% RSLogix 500 project Inventory_Management.RSS, saved by version 8.30.00.16 %
PROJECT "UNTITLED"    % processor: Bul.1763 MicroLogix 1100 Series B %

PROGRAM FILES
  LAD 2   9 rungs

DATA FILES
  O0 OUTPUT  4 elements
  I1 INPUT  6 elements
  S2 STATUS  66 elements
  B3 BINARY  1 elements
  T4 TIMER  1 elements
  C5 COUNTER  1 elements
  R6 CONTROL  1 elements
  N7 INTEGER  4 elements
  F8 FLOAT  1 elements
  ST9 STRING  10 elements

LADDER 2
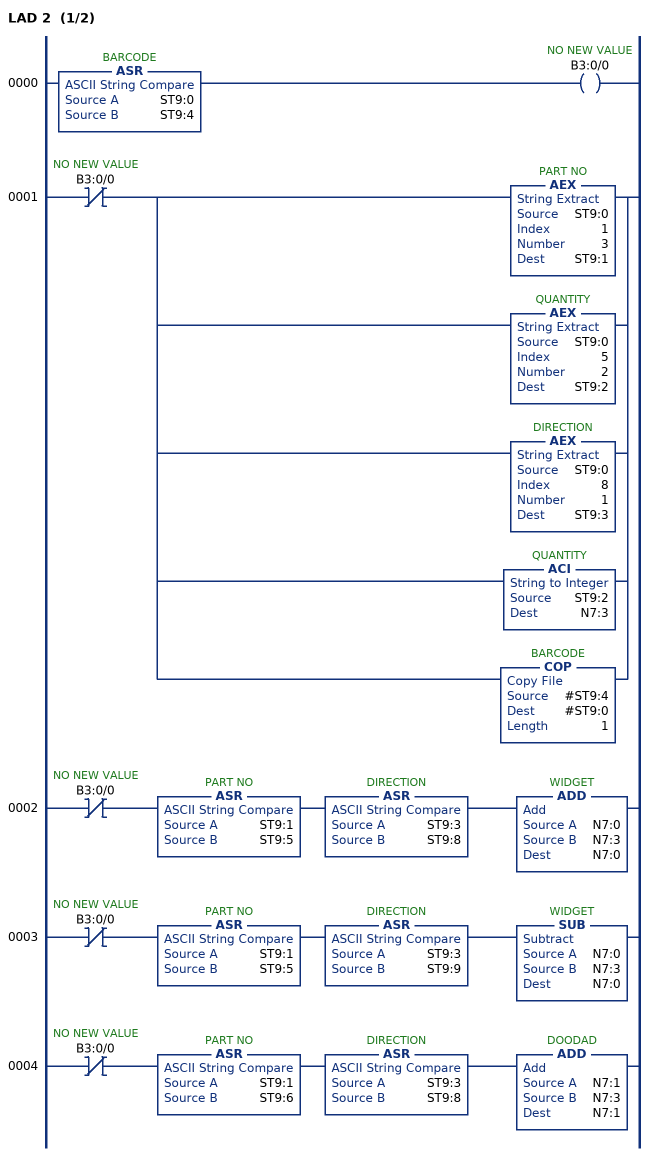
% Rung: 0 %
SOR ASR ST9:0 ST9:4 OTE B3:0/0 EOR
%   ST9:0  "BARCODE" %
%   B3:0/0  "NO NEW VALUE" %
% Rung: 1 %
SOR XIO B3:0/0 BST AEX ST9:0 1 3 ST9:1 NXB AEX ST9:0 5 2 ST9:2 NXB AEX ST9:0 8 1 ST9:3 NXB ACI ST9:2 N7:3 NXB COP #ST9:4 #ST9:0 1 BND EOR
%   B3:0/0  "NO NEW VALUE" %
%   ST9:0  "BARCODE" %
%   ST9:1  "PART NO" %
%   ST9:2  "QUANTITY" %
%   ST9:3  "DIRECTION" %
%   N7:3  "QUANTITY" %
% Rung: 2 %
SOR XIO B3:0/0 ASR ST9:1 ST9:5 ASR ST9:3 ST9:8 ADD N7:0 N7:3 N7:0 EOR
%   B3:0/0  "NO NEW VALUE" %
%   ST9:1  "PART NO" %
%   ST9:3  "DIRECTION" %
%   N7:0  "WIDGET" %
%   N7:3  "QUANTITY" %
% Rung: 3 %
SOR XIO B3:0/0 ASR ST9:1 ST9:5 ASR ST9:3 ST9:9 SUB N7:0 N7:3 N7:0 EOR
%   B3:0/0  "NO NEW VALUE" %
%   ST9:1  "PART NO" %
%   ST9:3  "DIRECTION" %
%   N7:0  "WIDGET" %
%   N7:3  "QUANTITY" %
% Rung: 4 %
SOR XIO B3:0/0 ASR ST9:1 ST9:6 ASR ST9:3 ST9:8 ADD N7:1 N7:3 N7:1 EOR
%   B3:0/0  "NO NEW VALUE" %
%   ST9:1  "PART NO" %
%   ST9:6  "PART NO" %
%   ST9:3  "DIRECTION" %
%   N7:1  "DOODAD" %
%   N7:3  "QUANTITY" %

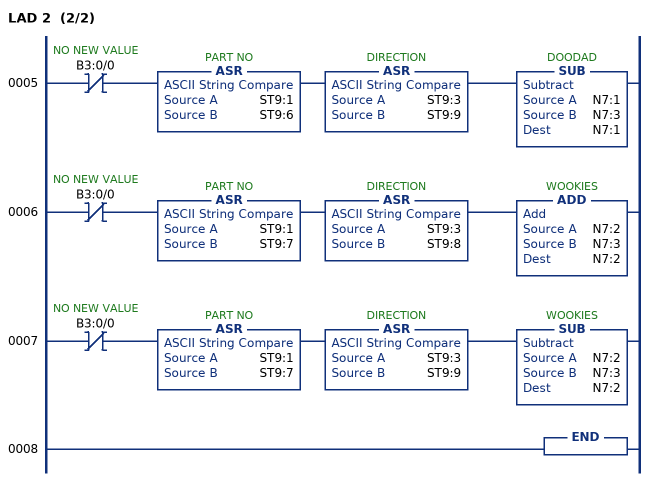
% Rung: 5 %
SOR XIO B3:0/0 ASR ST9:1 ST9:6 ASR ST9:3 ST9:9 SUB N7:1 N7:3 N7:1 EOR
%   B3:0/0  "NO NEW VALUE" %
%   ST9:1  "PART NO" %
%   ST9:6  "PART NO" %
%   ST9:3  "DIRECTION" %
%   N7:1  "DOODAD" %
%   N7:3  "QUANTITY" %
% Rung: 6 %
SOR XIO B3:0/0 ASR ST9:1 ST9:7 ASR ST9:3 ST9:8 ADD N7:2 N7:3 N7:2 EOR
%   B3:0/0  "NO NEW VALUE" %
%   ST9:1  "PART NO" %
%   ST9:3  "DIRECTION" %
%   N7:2  "WOOKIES" %
%   N7:3  "QUANTITY" %
% Rung: 7 %
SOR XIO B3:0/0 ASR ST9:1 ST9:7 ASR ST9:3 ST9:9 SUB N7:2 N7:3 N7:2 EOR
%   B3:0/0  "NO NEW VALUE" %
%   ST9:1  "PART NO" %
%   ST9:3  "DIRECTION" %
%   N7:2  "WOOKIES" %
%   N7:3  "QUANTITY" %
% Rung: 8 %
SOR END EOR

OTHER DOCUMENTED ADDRESSES
  ST0:0  "BARCODE SCAN"
  ST9:0.0  "BARCODE"
  ST9:1.0  "PART NO"
  ST9:2.0  "QUANTITY"
  ST9:3.0  "DIRECTION"
  ST9:4.0  "EMPTY STRING"
  ST9:5.0  "WIDGET"
  ST9:6.0  "DOODAD"
  ST9:7.0  "WOOKIES"

DATA TABLE (non-zero values as saved)
DATA B3
% B3:0 % 0X0001
DATA N7
% N7:0 % -18 -13 -18 1
DATA ST9
% ST9:1 % "149"
% ST9:2 % "1:"
% ST9:3 % "2"
% ST9:5 % "123"
% ST9:6 % "456"
% ST9:7 % "789"
% ST9:8 % "1"
% ST9:9 % "2"
